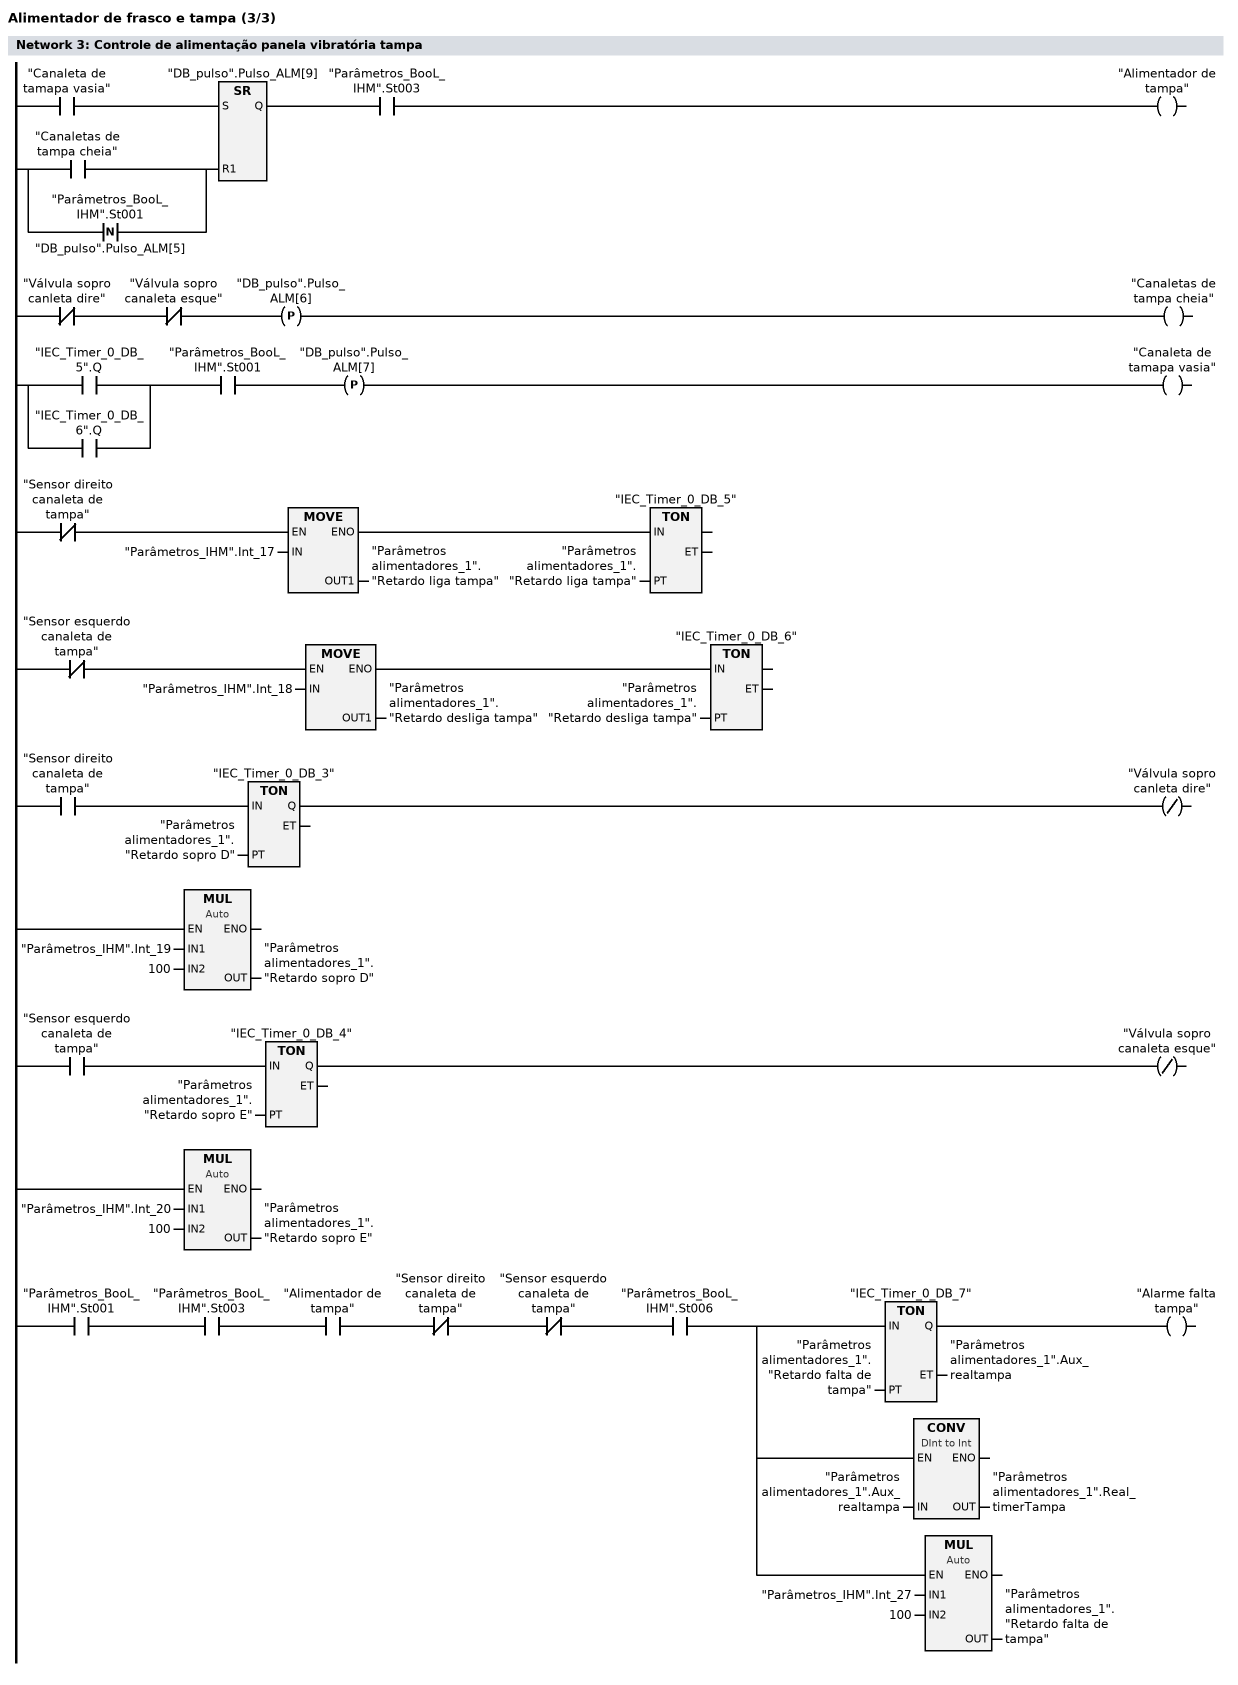
   #_w1 := NOT "Parâmetros_BooL_IHM".St001 AND "DB_pulso".Pulso_ALM[5];   // falling edge of "Parâmetros_BooL_IHM".St001
   "DB_pulso".Pulso_ALM[5] := "Parâmetros_BooL_IHM".St001;
   IF "Canaleta de tamapa vasia" THEN
       "DB_pulso".Pulso_ALM[9] := TRUE;   // SR flip-flop
   END_IF;
   IF "Canaletas de tampa cheia" OR #_w1 THEN "DB_pulso".Pulso_ALM[9] := FALSE; END_IF;
   "Alimentador de tampa" := "DB_pulso".Pulso_ALM[9] AND "Parâmetros_BooL_IHM".St003;
   #_w2 := NOT "Válvula sopro canleta dire" AND NOT "Válvula sopro canaleta esque";
   #_w3 := #_w2 AND NOT "DB_pulso".Pulso_ALM[6];   // rising edge
   "DB_pulso".Pulso_ALM[6] := #_w2;
   "Canaletas de tampa cheia" := #_w3;
   #_w4 := ("IEC_Timer_0_DB_5".Q OR "IEC_Timer_0_DB_6".Q) AND "Parâmetros_BooL_IHM".St001;
   #_w5 := #_w4 AND NOT "DB_pulso".Pulso_ALM[7];   // rising edge
   "DB_pulso".Pulso_ALM[7] := #_w4;
   "Canaleta de tamapa vasia" := #_w5;
   #_w6 := NOT "Sensor direito canaleta de tampa";
   IF #_w6 THEN "Parâmetros alimentadores_1"."Retardo liga tampa" := "Parâmetros_IHM".Int_17; END_IF;
   "IEC_Timer_0_DB_5".TON(IN := #_w6, PT := "Parâmetros alimentadores_1"."Retardo liga tampa");
   #_w7 := NOT "Sensor esquerdo canaleta de tampa";
   IF #_w7 THEN "Parâmetros alimentadores_1"."Retardo desliga tampa" := "Parâmetros_IHM".Int_18; END_IF;
   "IEC_Timer_0_DB_6".TON(IN := #_w7, PT := "Parâmetros alimentadores_1"."Retardo desliga tampa");
   "IEC_Timer_0_DB_3".TON(IN := "Sensor direito canaleta de tampa",
                          PT := "Parâmetros alimentadores_1"."Retardo sopro D");
   "Válvula sopro canleta dire" := NOT "IEC_Timer_0_DB_3".Q;
   "Parâmetros alimentadores_1"."Retardo sopro D" := "Parâmetros_IHM".Int_19 * 100;
   "IEC_Timer_0_DB_4".TON(IN := "Sensor esquerdo canaleta de tampa",
                          PT := "Parâmetros alimentadores_1"."Retardo sopro E");
   "Válvula sopro canaleta esque" := NOT "IEC_Timer_0_DB_4".Q;
   "Parâmetros alimentadores_1"."Retardo sopro E" := "Parâmetros_IHM".Int_20 * 100;
   #_w8 := "Parâmetros_BooL_IHM".St001 AND "Parâmetros_BooL_IHM".St003 AND "Alimentador de tampa" AND NOT "Sensor direito canaleta de tampa" AND NOT "Sensor esquerdo canaleta de tampa" AND "Parâmetros_BooL_IHM".St006;
   "IEC_Timer_0_DB_7".TON(IN := #_w8,
                          PT := "Parâmetros alimentadores_1"."Retardo falta de tampa",
                          ET => "Parâmetros alimentadores_1".Aux_realtampa);
   "Alarme falta tampa" := "IEC_Timer_0_DB_7".Q;
   IF #_w8 THEN
       "Parâmetros alimentadores_1".Real_timerTampa := DINT_TO_INT("Parâmetros alimentadores_1".Aux_realtampa);
       "Parâmetros alimentadores_1"."Retardo falta de tampa" := "Parâmetros_IHM".Int_27 * 100;
   END_IF;
END_REGION
END_FUNCTION

FUNCTION "Controle de produção" : Void   // FC7, LAD
{ S7_Optimized_Access := 'TRUE' }
VERSION : 0.1
   VAR_INPUT
      Habilita_contrle : Bool;
      Deslocamento_transmissão : Bool;
      Fim_envase : Bool;
      Sensor_detector : Bool;
      Rejeito : Bool;
   END_VAR
   VAR_OUTPUT
      Portão_rejeito : Bool;
      Pulso_inspeção : Bool;
   END_VAR
   VAR_IN_OUT
      Controle_habilitado : Bool;
      Total_produção : Int;
      Reprovado : Int;
      Peças_boas : Int;
      Setup_lote : Int;
   END_VAR
   VAR_TEMP   // added for the SCL form of the ladder/FBD networks
      _w1 : Bool;
      _w2 : Bool;
   END_VAR
BEGIN

REGION Network 1: Habilita controle de produção
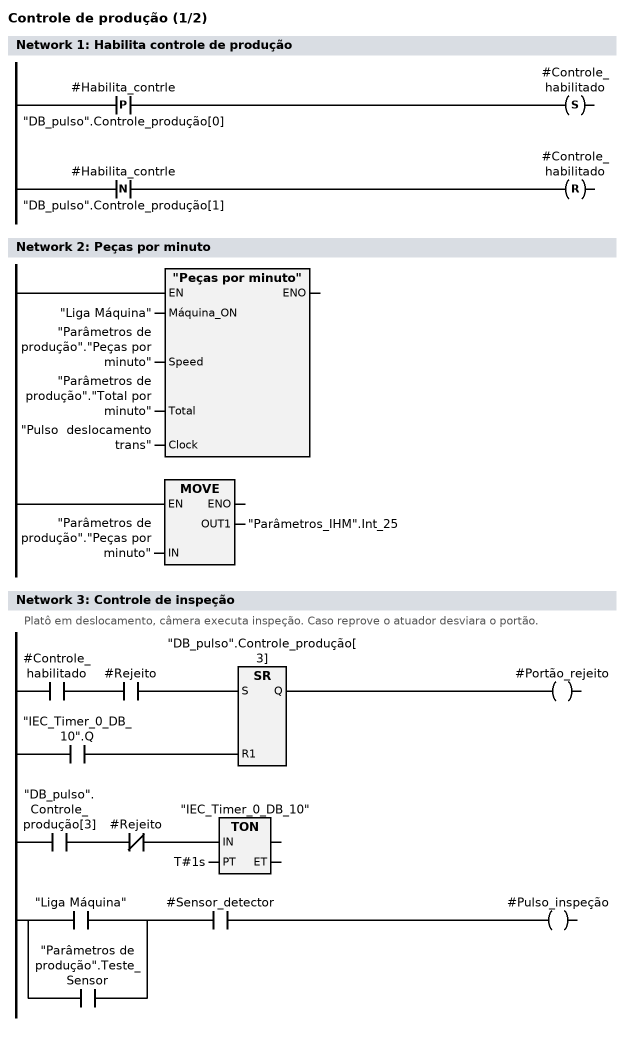
   RUNG wire#powerrail
      P_Contact(operand := #Habilita_contrle, bit := "DB_pulso".Controle_produção[0])
      S_Coil( #Controle_habilitado )
   END_RUNG
   RUNG wire#powerrail
      N_Contact(operand := #Habilita_contrle, bit := "DB_pulso".Controle_produção[1])
      R_Coil( #Controle_habilitado )
   END_RUNG
   // the same network as SCL:
   #_w1 := #Habilita_contrle AND NOT "DB_pulso".Controle_produção[0];   // rising edge of #Habilita_contrle
   "DB_pulso".Controle_produção[0] := #Habilita_contrle;
   IF #_w1 THEN #Controle_habilitado := TRUE; END_IF;
   #_w2 := NOT #Habilita_contrle AND "DB_pulso".Controle_produção[1];   // falling edge of #Habilita_contrle
   "DB_pulso".Controle_produção[1] := #Habilita_contrle;
   IF #_w2 THEN #Controle_habilitado := FALSE; END_IF;
END_REGION

REGION Network 2: Peças por minuto
   RUNG wire#powerrail
      "Peças por minuto"(Máquina_ON := "Liga Máquina", Speed := "Parâmetros de produção"."Peças por minuto", Total := "Parâmetros de produção"."Total por minuto", Clock := "Pulso  deslocamento trans")
   END_RUNG
   RUNG wire#powerrail
      Move(in := "Parâmetros de produção"."Peças por minuto", out1 => "Parâmetros_IHM".Int_25)
   END_RUNG
   // the same network as SCL:
   "Peças por minuto"(Máquina_ON := "Liga Máquina",
                      Speed := "Parâmetros de produção"."Peças por minuto",
                      Total := "Parâmetros de produção"."Total por minuto",
                      Clock := "Pulso  deslocamento trans");
   "Parâmetros_IHM".Int_25 := "Parâmetros de produção"."Peças por minuto";
END_REGION

REGION Network 3: Controle de inspeção
   // Platô em deslocamento, câmera executa inspeção. Caso reprove o atuador desviara o portão.
   IF #Controle_habilitado AND #Rejeito THEN
       "DB_pulso".Controle_produção[3] := TRUE;   // SR flip-flop
   END_IF;
   IF "IEC_Timer_0_DB_10".Q THEN "DB_pulso".Controle_produção[3] := FALSE; END_IF;
   #Portão_rejeito := "DB_pulso".Controle_produção[3];
   "IEC_Timer_0_DB_10".TON(IN := "DB_pulso".Controle_produção[3] AND NOT #Rejeito, PT := T#1s);
   #Pulso_inspeção := ("Liga Máquina" OR "Parâmetros de produção".Teste_Sensor) AND #Sensor_detector;
END_REGION

REGION Network 4: Contagem de produção
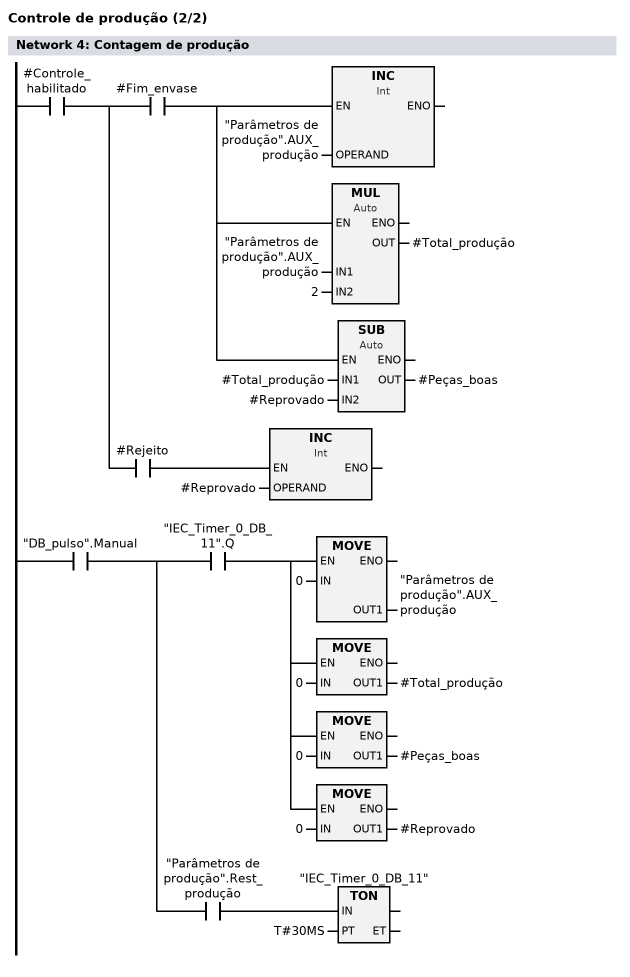
   IF #Controle_habilitado AND #Fim_envase THEN
       "Parâmetros de produção".AUX_produção := "Parâmetros de produção".AUX_produção + 1;
       #Total_produção := "Parâmetros de produção".AUX_produção * 2;
       #Peças_boas := #Total_produção - #Reprovado;
   END_IF;
   IF #Controle_habilitado AND #Rejeito THEN #Reprovado := #Reprovado + 1; END_IF;
   IF "DB_pulso".Manual AND "IEC_Timer_0_DB_11".Q THEN
       "Parâmetros de produção".AUX_produção := 0;
       #Total_produção := 0;
       #Peças_boas := 0;
       #Reprovado := 0;
   END_IF;
   "IEC_Timer_0_DB_11".TON(IN := "DB_pulso".Manual AND "Parâmetros de produção".Rest_produção, PT := T#30MS);
END_REGION
END_FUNCTION

FUNCTION "Alarme" : Void   // FC8, LAD
{ S7_Optimized_Access := 'TRUE' }
VERSION : 0.1
   VAR_OUTPUT
      Restfalahaservodrives : Bool;
      Falha_sincronismo : Bool;
      Atenção : Bool;
   END_VAR
   VAR_IN_OUT
      Status_sincronismo : Bool;
   END_VAR
   VAR_TEMP
      Reset1 : Bool;
      reset2 : Bool;
      reset3 : Bool;
      Status_sincornismo : Bool;
   END_VAR
   VAR_TEMP   // added for the SCL form of the ladder/FBD networks
      _w1 : Bool;
      _w2 : Bool;
      _w3 : Bool;
      _w4 : Bool;
   END_VAR
BEGIN

REGION Network 1: Alarme ativo
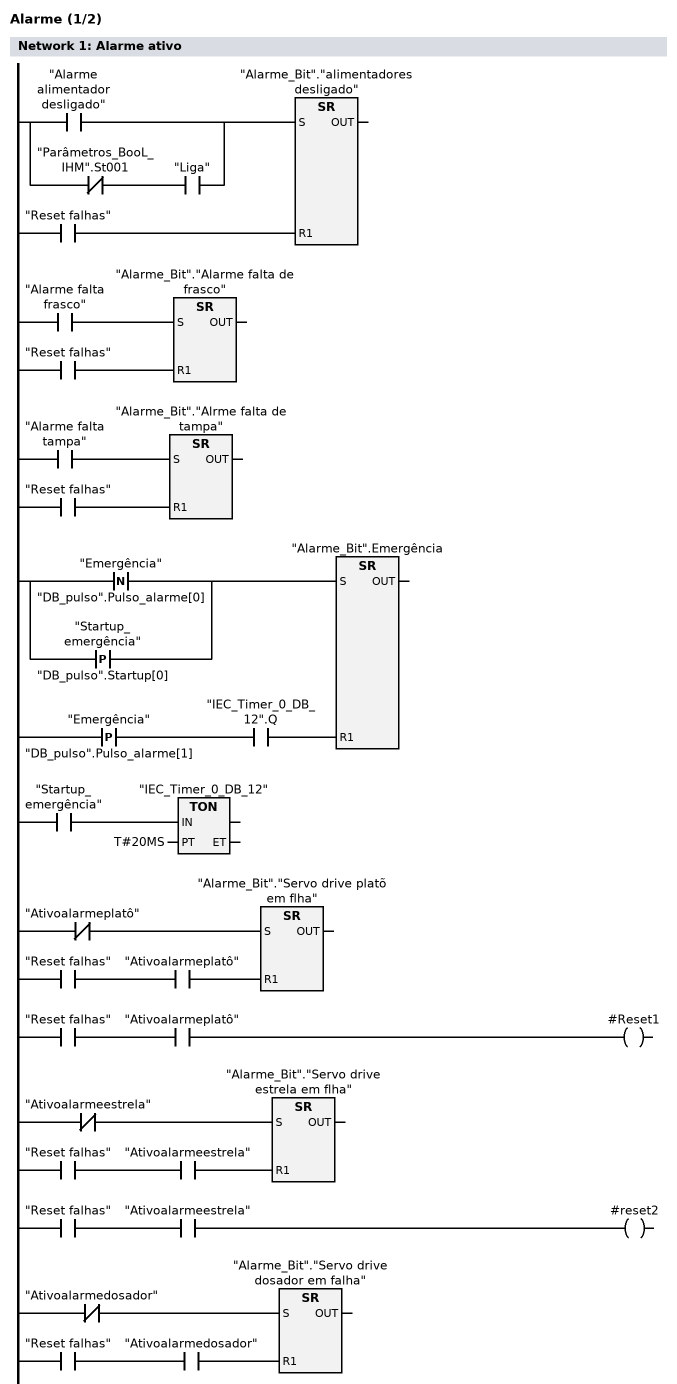
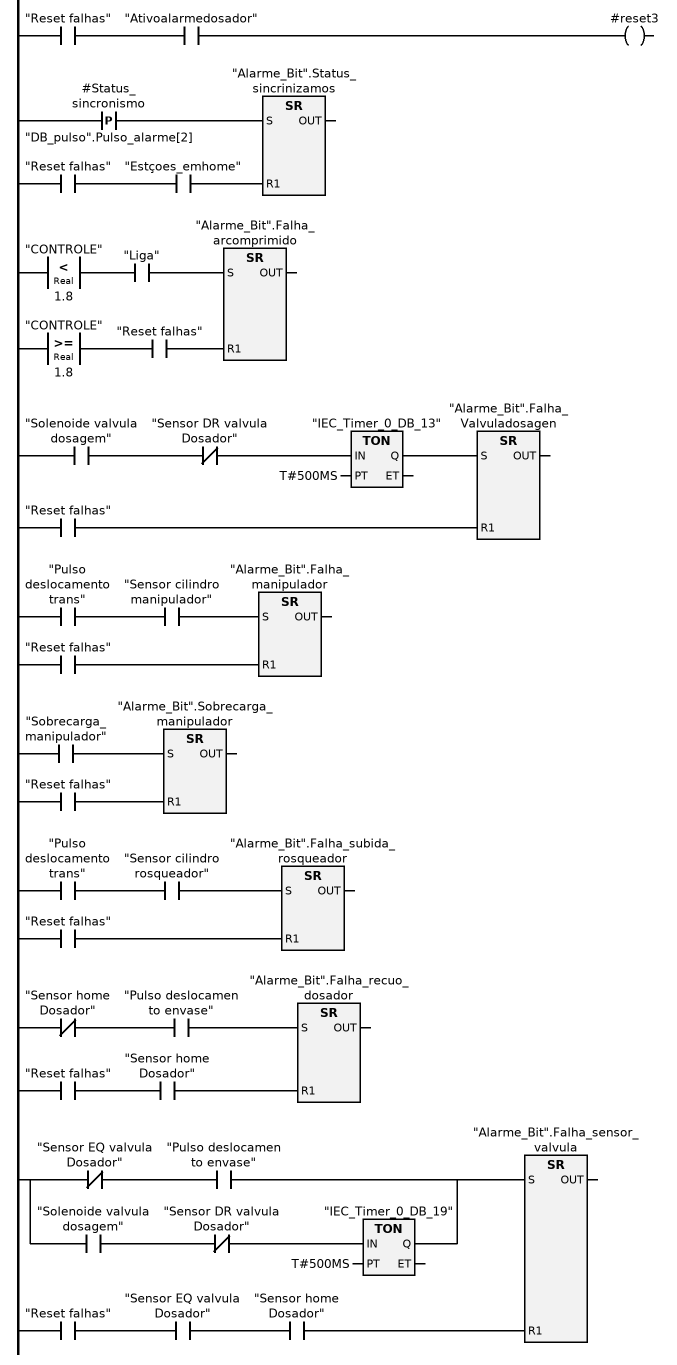
   IF "Alarme alimentador desligado" OR (NOT "Parâmetros_BooL_IHM".St001 AND "Liga") THEN
       "Alarme_Bit"."alimentadores desligado" := TRUE;   // SR flip-flop
   END_IF;
   IF "Reset falhas" THEN "Alarme_Bit"."alimentadores desligado" := FALSE; END_IF;
   IF "Alarme falta frasco" THEN
       "Alarme_Bit"."Alarme falta de frasco" := TRUE;   // SR flip-flop
   END_IF;
   IF "Reset falhas" THEN "Alarme_Bit"."Alarme falta de frasco" := FALSE; END_IF;
   IF "Alarme falta tampa" THEN
       "Alarme_Bit"."Alrme falta de tampa" := TRUE;   // SR flip-flop
   END_IF;
   IF "Reset falhas" THEN "Alarme_Bit"."Alrme falta de tampa" := FALSE; END_IF;
   #_w1 := NOT "Emergência" AND "DB_pulso".Pulso_alarme[0];   // falling edge of "Emergência"
   "DB_pulso".Pulso_alarme[0] := "Emergência";
   #_w2 := "Startup_emergência" AND NOT "DB_pulso".Startup[0];   // rising edge of "Startup_emergência"
   "DB_pulso".Startup[0] := "Startup_emergência";
   #_w3 := "Emergência" AND NOT "DB_pulso".Pulso_alarme[1];   // rising edge of "Emergência"
   "DB_pulso".Pulso_alarme[1] := "Emergência";
   IF #_w1 OR #_w2 THEN
       "Alarme_Bit".Emergência := TRUE;   // SR flip-flop
   END_IF;
   IF #_w3 AND "IEC_Timer_0_DB_12".Q THEN "Alarme_Bit".Emergência := FALSE; END_IF;
   "IEC_Timer_0_DB_12".TON(IN := "Startup_emergência", PT := T#20MS);
   IF NOT "Ativoalarmeplatô" THEN
       "Alarme_Bit"."Servo drive platõ em flha" := TRUE;   // SR flip-flop
   END_IF;
   IF "Reset falhas" AND "Ativoalarmeplatô" THEN "Alarme_Bit"."Servo drive platõ em flha" := FALSE; END_IF;
   #Reset1 := "Reset falhas" AND "Ativoalarmeplatô";
   IF NOT "Ativoalarmeestrela" THEN
       "Alarme_Bit"."Servo drive estrela em flha" := TRUE;   // SR flip-flop
   END_IF;
   IF "Reset falhas" AND "Ativoalarmeestrela" THEN
       "Alarme_Bit"."Servo drive estrela em flha" := FALSE;
   END_IF;
   #reset2 := "Reset falhas" AND "Ativoalarmeestrela";
   IF NOT "Ativoalarmedosador" THEN
       "Alarme_Bit"."Servo drive dosador em falha" := TRUE;   // SR flip-flop
   END_IF;
   IF "Reset falhas" AND "Ativoalarmedosador" THEN
       "Alarme_Bit"."Servo drive dosador em falha" := FALSE;
   END_IF;
   #reset3 := "Reset falhas" AND "Ativoalarmedosador";
   #_w4 := #Status_sincronismo AND NOT "DB_pulso".Pulso_alarme[2];   // rising edge of #Status_sincronismo
   "DB_pulso".Pulso_alarme[2] := #Status_sincronismo;
   IF #_w4 THEN
       "Alarme_Bit".Status_sincrinizamos := TRUE;   // SR flip-flop
   END_IF;
   IF "Reset falhas" AND "Estçoes_emhome" THEN "Alarme_Bit".Status_sincrinizamos := FALSE; END_IF;
   IF ("CONTROLE" < 1.8) AND "Liga" THEN
       "Alarme_Bit".Falha_arcomprimido := TRUE;   // SR flip-flop
   END_IF;
   IF ("CONTROLE" >= 1.8) AND "Reset falhas" THEN "Alarme_Bit".Falha_arcomprimido := FALSE; END_IF;
   "IEC_Timer_0_DB_13".TON(IN := "Solenoide valvula dosagem" AND NOT "Sensor DR valvula Dosador", PT := T#500MS);
   IF "IEC_Timer_0_DB_13".Q THEN
       "Alarme_Bit".Falha_Valvuladosagen := TRUE;   // SR flip-flop
   END_IF;
   IF "Reset falhas" THEN "Alarme_Bit".Falha_Valvuladosagen := FALSE; END_IF;
   IF "Pulso  deslocamento trans" AND "Sensor cilindro manipulador" THEN
       "Alarme_Bit".Falha_manipulador := TRUE;   // SR flip-flop
   END_IF;
   IF "Reset falhas" THEN "Alarme_Bit".Falha_manipulador := FALSE; END_IF;
   IF "Sobrecarga_manipulador" THEN
       "Alarme_Bit".Sobrecarga_manipulador := TRUE;   // SR flip-flop
   END_IF;
   IF "Reset falhas" THEN "Alarme_Bit".Sobrecarga_manipulador := FALSE; END_IF;
   IF "Pulso  deslocamento trans" AND "Sensor cilindro rosqueador" THEN
       "Alarme_Bit".Falha_subida_rosqueador := TRUE;   // SR flip-flop
   END_IF;
   IF "Reset falhas" THEN "Alarme_Bit".Falha_subida_rosqueador := FALSE; END_IF;
   IF NOT "Sensor home Dosador" AND "Pulso deslocamento envase" THEN
       "Alarme_Bit".Falha_recuo_dosador := TRUE;   // SR flip-flop
   END_IF;
   IF "Reset falhas" AND "Sensor home Dosador" THEN "Alarme_Bit".Falha_recuo_dosador := FALSE; END_IF;
   "IEC_Timer_0_DB_19".TON(IN := "Solenoide valvula dosagem" AND NOT "Sensor DR valvula Dosador", PT := T#500MS);
   IF (NOT "Sensor EQ valvula Dosador" AND "Pulso deslocamento envase") OR "IEC_Timer_0_DB_19".Q THEN
       "Alarme_Bit".Falha_sensor_valvula := TRUE;   // SR flip-flop
   END_IF;
   IF "Reset falhas" AND "Sensor EQ valvula Dosador" AND "Sensor home Dosador" THEN
       "Alarme_Bit".Falha_sensor_valvula := FALSE;
   END_IF;
END_REGION

REGION Network 2: Reset alarme servo drives
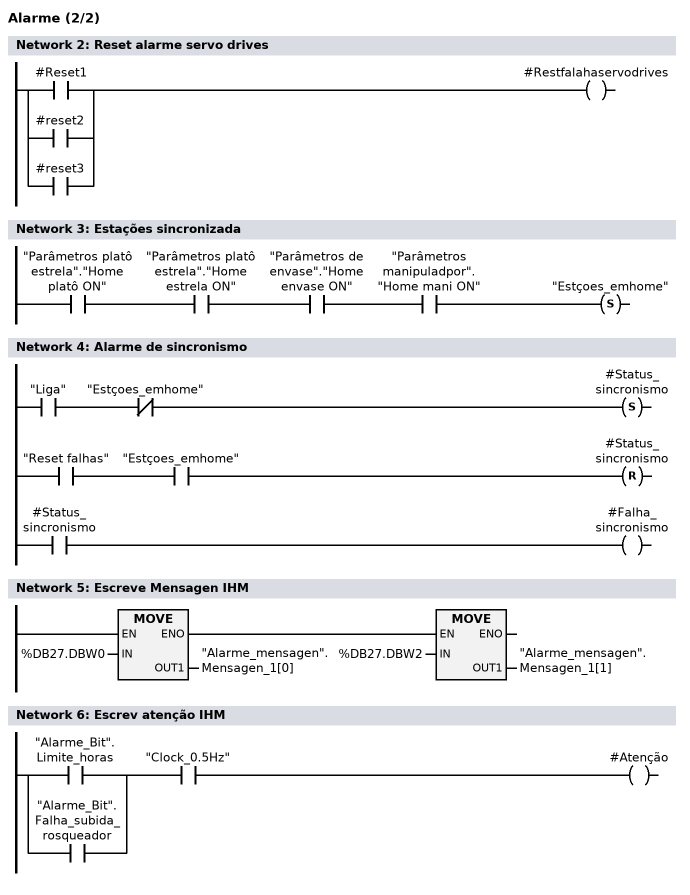
   RUNG wire#powerrail
      Contact( #Reset1 )
      wire#w1
      Coil( #Restfalahaservodrives )
   END_RUNG
   RUNG wire#powerrail
      Contact( #reset2 )
   END_RUNG wire#w1
   RUNG wire#powerrail
      Contact( #reset3 )
   END_RUNG wire#w1
   // the same network as SCL:
   #Restfalahaservodrives := #Reset1 OR #reset2 OR #reset3;
END_REGION

REGION Network 3: Estações sincronizada
   RUNG wire#powerrail
      Contact( "Parâmetros platô estrela"."Home platô ON" )
      Contact( "Parâmetros platô estrela"."Home estrela ON" )
      Contact( "Parâmetros de envase"."Home envase ON" )
      Contact( "Parâmetros manipuladpor"."Home mani ON" )
      S_Coil( "Estçoes_emhome" )
   END_RUNG
   // the same network as SCL:
   IF "Parâmetros platô estrela"."Home platô ON" AND "Parâmetros platô estrela"."Home estrela ON" AND "Parâmetros de envase"."Home envase ON" AND "Parâmetros manipuladpor"."Home mani ON" THEN
       "Estçoes_emhome" := TRUE;
   END_IF;
END_REGION

REGION Network 4: Alarme de sincronismo
   RUNG wire#powerrail
      Contact( "Liga" )
      I_Contact( "Estçoes_emhome" )
      S_Coil( #Status_sincronismo )
   END_RUNG
   RUNG wire#powerrail
      Contact( "Reset falhas" )
      Contact( "Estçoes_emhome" )
      R_Coil( #Status_sincronismo )
   END_RUNG
   RUNG wire#powerrail
      Contact( #Status_sincronismo )
      Coil( #Falha_sincronismo )
   END_RUNG
   // the same network as SCL:
   IF "Liga" AND NOT "Estçoes_emhome" THEN #Status_sincronismo := TRUE; END_IF;
   IF "Reset falhas" AND "Estçoes_emhome" THEN #Status_sincronismo := FALSE; END_IF;
   #Falha_sincronismo := #Status_sincronismo;
END_REGION

REGION Network 5: Escreve Mensagen IHM
   RUNG wire#powerrail
      Move(in := %DB27.DBW0, out1 => "Alarme_mensagen".Mensagen_1[0])
      Move(in := %DB27.DBW2, out1 => "Alarme_mensagen".Mensagen_1[1])
   END_RUNG
   // the same network as SCL:
   "Alarme_mensagen".Mensagen_1[0] := %DB27.DBW0;
   "Alarme_mensagen".Mensagen_1[1] := %DB27.DBW2;
END_REGION

REGION Network 6: Escrev atenção IHM
   RUNG wire#powerrail
      Contact( "Alarme_Bit".Limite_horas )
      wire#w1
      Contact( "Clock_0.5Hz" )
      Coil( #Atenção )
   END_RUNG
   RUNG wire#powerrail
      Contact( "Alarme_Bit".Falha_subida_rosqueador )
   END_RUNG wire#w1
   // the same network as SCL:
   #Atenção := ("Alarme_Bit".Limite_horas OR "Alarme_Bit".Falha_subida_rosqueador) AND "Clock_0.5Hz";
END_REGION
END_FUNCTION

FUNCTION "AR Comprimido" : Void   // FC9, LAD
{ S7_Optimized_Access := 'TRUE' }
VERSION : 0.1
BEGIN

REGION Network 1: Leitura de sensor de pressão
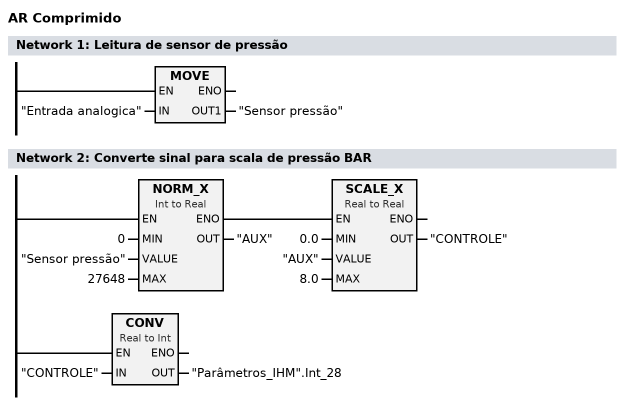
   RUNG wire#powerrail
      Move(in := "Entrada analogica", out1 => "Sensor pressão")
   END_RUNG
   // the same network as SCL:
   "Sensor pressão" := "Entrada analogica";
END_REGION

REGION Network 2: Converte sinal para scala de pressão BAR
   RUNG wire#powerrail
      { S7_Templates := "[SrcType := Int, DestType := Real]" } Normalize(min := 0, value := "Sensor pressão", max := 27648, out => "AUX")
      { S7_Templates := "[SrcType := Real, DestType := Real]" } Scale(min := 0.0, value := "AUX", max := 8.0, out => "CONTROLE")
   END_RUNG
   RUNG wire#powerrail
      { S7_Templates := "[SrcType := Real, DestType := Int]" } Convert(in := "CONTROLE", out => "Parâmetros_IHM".Int_28)
   END_RUNG
   // the same network as SCL:
   "AUX" := NORM_X(MIN := 0, VALUE := "Sensor pressão", MAX := 27648);
   "CONTROLE" := SCALE_X(MIN := 0.0, VALUE := "AUX", MAX := 8.0);
   "Parâmetros_IHM".Int_28 := REAL_TO_INT("CONTROLE");
END_REGION
END_FUNCTION

FUNCTION "Peças por minuto" : Void   // FC10, LAD
{ S7_Optimized_Access := 'TRUE' }
VERSION : 0.1
   VAR_INPUT
      Máquina_ON : Bool;
   END_VAR
   VAR_IN_OUT
      Speed : DInt;
      Total : DInt;
      Clock : Bool;
   END_VAR
BEGIN

REGION Network 1: Contador de peça por minuto
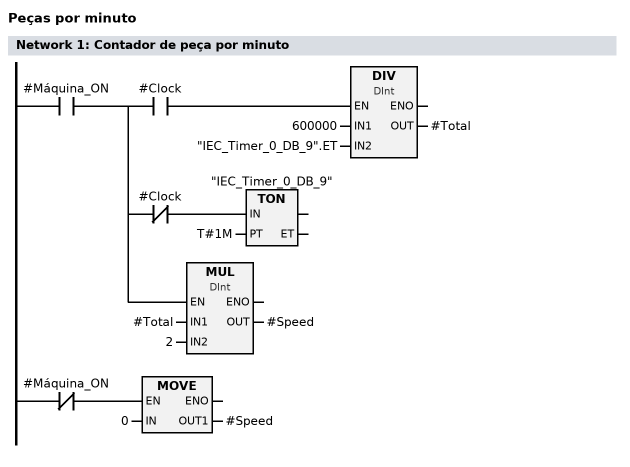
   IF #Máquina_ON AND #Clock THEN #Total := 600000 / "IEC_Timer_0_DB_9".ET; END_IF;
   "IEC_Timer_0_DB_9".TON(IN := #Máquina_ON AND NOT #Clock, PT := T#1M);
   IF #Máquina_ON THEN #Speed := #Total * 2; END_IF;
   IF NOT #Máquina_ON THEN #Speed := 0; END_IF;
END_REGION
END_FUNCTION

FUNCTION "Recipe" : Void   // FC11, LAD
{ S7_Optimized_Access := 'TRUE' }
VERSION : 0.1
   VAR_TEMP   // added for the SCL form of the ladder/FBD networks
      _w1 : Bool;
   END_VAR
BEGIN

REGION Network 1: Download recita
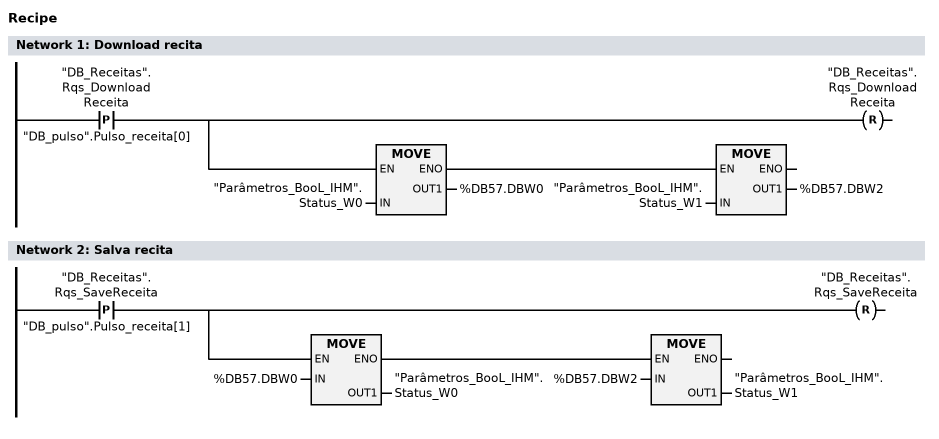
   RUNG wire#powerrail
      P_Contact(operand := "DB_Receitas".Rqs_DownloadReceita, bit := "DB_pulso".Pulso_receita[0])
      wire#w1
      R_Coil( "DB_Receitas".Rqs_DownloadReceita )
   END_RUNG
   RUNG wire#w1
      Move(in := "Parâmetros_BooL_IHM".Status_W0, out1 => %DB57.DBW0)
      Move(in := "Parâmetros_BooL_IHM".Status_W1, out1 => %DB57.DBW2)
   END_RUNG
   // the same network as SCL:
   #_w1 := "DB_Receitas".Rqs_DownloadReceita AND NOT "DB_pulso".Pulso_receita[0];   // rising edge of "DB_Receitas".Rqs_DownloadReceita
   "DB_pulso".Pulso_receita[0] := "DB_Receitas".Rqs_DownloadReceita;
   IF #_w1 THEN
       "DB_Receitas".Rqs_DownloadReceita := FALSE;
       %DB57.DBW0 := "Parâmetros_BooL_IHM".Status_W0;
       %DB57.DBW2 := "Parâmetros_BooL_IHM".Status_W1;
   END_IF;
END_REGION

REGION Network 2: Salva recita
   RUNG wire#powerrail
      P_Contact(operand := "DB_Receitas".Rqs_SaveReceita, bit := "DB_pulso".Pulso_receita[1])
      wire#w1
      R_Coil( "DB_Receitas".Rqs_SaveReceita )
   END_RUNG
   RUNG wire#w1
      Move(in := %DB57.DBW0, out1 => "Parâmetros_BooL_IHM".Status_W0)
      Move(in := %DB57.DBW2, out1 => "Parâmetros_BooL_IHM".Status_W1)
   END_RUNG
   // the same network as SCL:
   #_w1 := "DB_Receitas".Rqs_SaveReceita AND NOT "DB_pulso".Pulso_receita[1];   // rising edge of "DB_Receitas".Rqs_SaveReceita
   "DB_pulso".Pulso_receita[1] := "DB_Receitas".Rqs_SaveReceita;
   IF #_w1 THEN
       "DB_Receitas".Rqs_SaveReceita := FALSE;
       "Parâmetros_BooL_IHM".Status_W0 := %DB57.DBW0;
       "Parâmetros_BooL_IHM".Status_W1 := %DB57.DBW2;
   END_IF;
END_REGION
END_FUNCTION

FUNCTION "Habilita_estações" : Void   // FC12, LAD
{ S7_Optimized_Access := 'TRUE' }
VERSION : 0.1
BEGIN

REGION Network 1: ON OFF estações
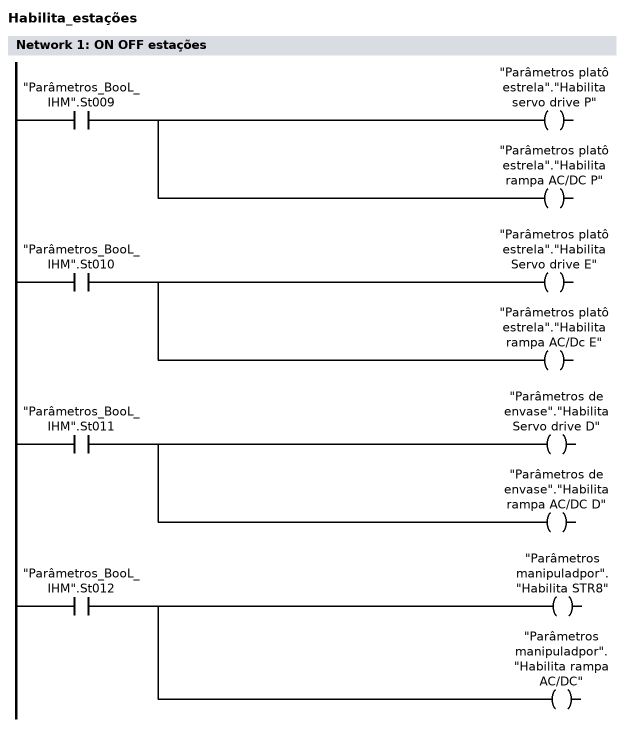
   RUNG wire#powerrail
      Contact( "Parâmetros_BooL_IHM".St009 )
      wire#w1
      Coil( "Parâmetros platô estrela"."Habilita servo drive P" )
   END_RUNG
   RUNG wire#w1
      Coil( "Parâmetros platô estrela"."Habilita rampa AC/DC P" )
   END_RUNG
   RUNG wire#powerrail
      Contact( "Parâmetros_BooL_IHM".St010 )
      wire#w2
      Coil( "Parâmetros platô estrela"."Habilita Servo drive E" )
   END_RUNG
   RUNG wire#w2
      Coil( "Parâmetros platô estrela"."Habilita rampa AC/Dc E" )
   END_RUNG
   RUNG wire#powerrail
      Contact( "Parâmetros_BooL_IHM".St011 )
      wire#w3
      Coil( "Parâmetros de envase"."Habilita Servo drive D" )
   END_RUNG
   RUNG wire#w3
      Coil( "Parâmetros de envase"."Habilita rampa AC/DC D" )
   END_RUNG
   RUNG wire#powerrail
      Contact( "Parâmetros_BooL_IHM".St012 )
      wire#w4
      Coil( "Parâmetros manipuladpor"."Habilita STR8" )
   END_RUNG
   RUNG wire#w4
      Coil( "Parâmetros manipuladpor"."Habilita rampa AC/DC" )
   END_RUNG
   // the same network as SCL:
   "Parâmetros platô estrela"."Habilita servo drive P" := "Parâmetros_BooL_IHM".St009;
   "Parâmetros platô estrela"."Habilita rampa AC/DC P" := "Parâmetros_BooL_IHM".St009;
   "Parâmetros platô estrela"."Habilita Servo drive E" := "Parâmetros_BooL_IHM".St010;
   "Parâmetros platô estrela"."Habilita rampa AC/Dc E" := "Parâmetros_BooL_IHM".St010;
   "Parâmetros de envase"."Habilita Servo drive D" := "Parâmetros_BooL_IHM".St011;
   "Parâmetros de envase"."Habilita rampa AC/DC D" := "Parâmetros_BooL_IHM".St011;
   "Parâmetros manipuladpor"."Habilita STR8" := "Parâmetros_BooL_IHM".St012;
   "Parâmetros manipuladpor"."Habilita rampa AC/DC" := "Parâmetros_BooL_IHM".St012;
END_REGION
END_FUNCTION

ORGANIZATION_BLOCK "Main"   // OB1, LAD, ProgramCycle
TITLE = "Main Program Sweep (Cycle)"
{ S7_Optimized_Access := 'TRUE' }
VERSION : 0.1
   VAR_INPUT
      Initial_Call : Bool;   // Initial call of this OB
      Remanence : Bool;   // =True, if remanent data are available
   END_VAR
   VAR_TEMP   // added for the SCL form of the ladder/FBD networks
      _w1 : Bool;
      _w2 : Bool;
      _w3 : Bool;
   END_VAR
BEGIN

REGION Network 1: Liga máquina
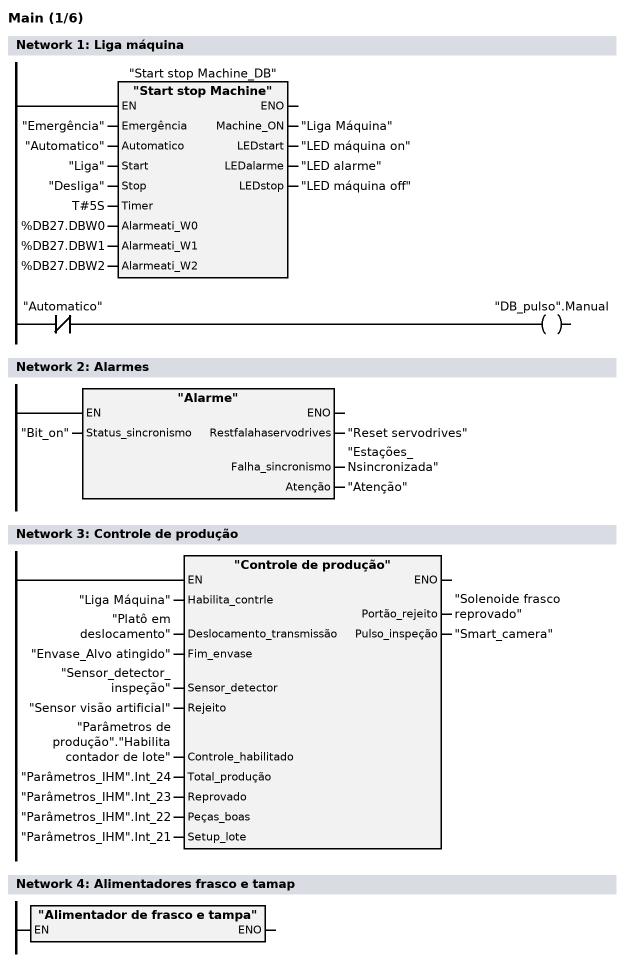
   RUNG wire#powerrail
      "Start stop Machine_DB"(Emergência := "Emergência", Automatico := "Automatico", Start := "Liga", Stop := "Desliga", "Timer" := T#5S, Alarmeati_W0 := %DB27.DBW0, Alarmeati_W1 := %DB27.DBW1, Alarmeati_W2 := %DB27.DBW2, Machine_ON => "Liga Máquina", LEDstart => "LED máquina on", LEDalarme => "LED alarme", LEDstop => "LED máquina off")
   END_RUNG
   RUNG wire#powerrail
      I_Contact( "Automatico" )
      Coil( "DB_pulso".Manual )
   END_RUNG
   // the same network as SCL:
   "Start stop Machine_DB"(Emergência := "Emergência",   // "Start stop Machine"
                           Automatico := "Automatico",
                           Start := "Liga",
                           Stop := "Desliga",
                           "Timer" := T#5S,
                           Alarmeati_W0 := %DB27.DBW0,
                           Alarmeati_W1 := %DB27.DBW1,
                           Alarmeati_W2 := %DB27.DBW2,
                           Machine_ON => "Liga Máquina",
                           LEDstart => "LED máquina on",
                           LEDalarme => "LED alarme",
                           LEDstop => "LED máquina off");
   "DB_pulso".Manual := NOT "Automatico";
END_REGION

REGION Network 2: Alarmes
   RUNG wire#powerrail
      "Alarme"(Status_sincronismo := "Bit_on", Restfalahaservodrives => "Reset servodrives", Falha_sincronismo => "Estações_Nsincronizada", Atenção => "Atenção")
   END_RUNG
   // the same network as SCL:
   "Alarme"(Status_sincronismo := "Bit_on",
            Restfalahaservodrives => "Reset servodrives",
            Falha_sincronismo => "Estações_Nsincronizada",
            Atenção => "Atenção");
END_REGION

REGION Network 3: Controle de produção
   RUNG wire#powerrail
      "Controle de produção"(Habilita_contrle := "Liga Máquina", Deslocamento_transmissão := "Platô em deslocamento", Fim_envase := "Envase_Alvo atingido", Sensor_detector := "Sensor_detector_inspeção", Rejeito := "Sensor visão artificial", Controle_habilitado := "Parâmetros de produção"."Habilita contador de lote", Total_produção := "Parâmetros_IHM".Int_24, Reprovado := "Parâmetros_IHM".Int_23, Peças_boas := "Parâmetros_IHM".Int_22, Setup_lote := "Parâmetros_IHM".Int_21, Portão_rejeito => "Solenoide frasco reprovado", Pulso_inspeção => "Smart_camera")
   END_RUNG
   // the same network as SCL:
   "Controle de produção"(Habilita_contrle := "Liga Máquina",
                          Deslocamento_transmissão := "Platô em deslocamento",
                          Fim_envase := "Envase_Alvo atingido",
                          Sensor_detector := "Sensor_detector_inspeção",
                          Rejeito := "Sensor visão artificial",
                          Controle_habilitado := "Parâmetros de produção"."Habilita contador de lote",
                          Total_produção := "Parâmetros_IHM".Int_24,
                          Reprovado := "Parâmetros_IHM".Int_23,
                          Peças_boas := "Parâmetros_IHM".Int_22,
                          Setup_lote := "Parâmetros_IHM".Int_21,
                          Portão_rejeito => "Solenoide frasco reprovado",
                          Pulso_inspeção => "Smart_camera");
END_REGION

REGION Network 4: Alimentadores frasco e tamap
   RUNG wire#powerrail
      "Alimentador de frasco e tampa"()
   END_RUNG
   // the same network as SCL:
   "Alimentador de frasco e tampa"();
END_REGION

REGION Network 5: Transmissão Plato e estrela
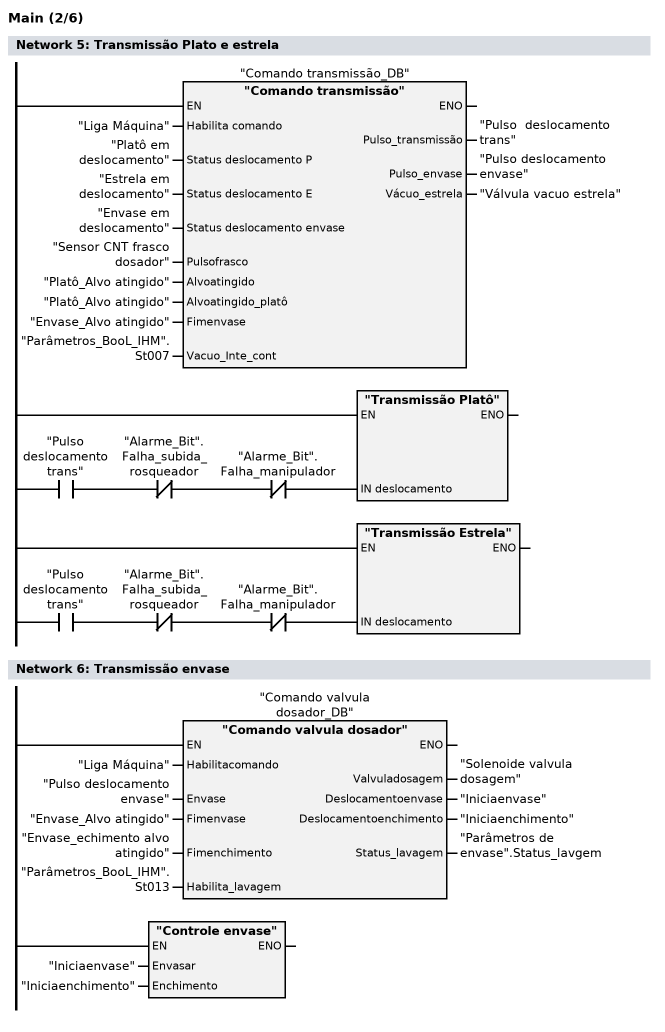
   RUNG wire#powerrail
      "Comando transmissão_DB"("Habilita comando" := "Liga Máquina", "Status deslocamento P" := "Platô em deslocamento", "Status deslocamento E" := "Estrela em deslocamento", "Status deslocamento envase" := "Envase em deslocamento", Pulsofrasco := "Sensor CNT frasco dosador", Alvoatingido := "Platô_Alvo atingido", Alvoatingido_platô := "Platô_Alvo atingido", Fimenvase := "Envase_Alvo atingido", Vacuo_Inte_cont := "Parâmetros_BooL_IHM".St007, Pulso_transmissão => "Pulso  deslocamento trans", Pulso_envase => "Pulso deslocamento envase", Vácuo_estrela => "Válvula vacuo estrela")
   END_RUNG
   RUNG wire#powerrail
      "Transmissão Platô"("IN deslocamento" := wire#w1)
   END_RUNG
   RUNG wire#powerrail
      Contact( "Pulso  deslocamento trans" )
      I_Contact( "Alarme_Bit".Falha_subida_rosqueador )
      I_Contact( "Alarme_Bit".Falha_manipulador )
   END_RUNG wire#w1
   RUNG wire#powerrail
      "Transmissão Estrela"("IN deslocamento" := wire#w2)
   END_RUNG
   RUNG wire#powerrail
      Contact( "Pulso  deslocamento trans" )
      I_Contact( "Alarme_Bit".Falha_subida_rosqueador )
      I_Contact( "Alarme_Bit".Falha_manipulador )
   END_RUNG wire#w2
   // the same network as SCL:
   "Comando transmissão_DB"("Habilita comando" := "Liga Máquina",   // "Comando transmissão"
                           "Status deslocamento P" := "Platô em deslocamento",
                           "Status deslocamento E" := "Estrela em deslocamento",
                           "Status deslocamento envase" := "Envase em deslocamento",
                           Pulsofrasco := "Sensor CNT frasco dosador",
                           Alvoatingido := "Platô_Alvo atingido",
                           Alvoatingido_platô := "Platô_Alvo atingido",
                           Fimenvase := "Envase_Alvo atingido",
                           Vacuo_Inte_cont := "Parâmetros_BooL_IHM".St007,
                           Pulso_transmissão => "Pulso  deslocamento trans",
                           Pulso_envase => "Pulso deslocamento envase",
                           Vácuo_estrela => "Válvula vacuo estrela");
   "Transmissão Platô"("IN deslocamento" := "Pulso  deslocamento trans" AND NOT "Alarme_Bit".Falha_subida_rosqueador AND NOT "Alarme_Bit".Falha_manipulador);
   "Transmissão Estrela"("IN deslocamento" := "Pulso  deslocamento trans" AND NOT "Alarme_Bit".Falha_subida_rosqueador AND NOT "Alarme_Bit".Falha_manipulador);
END_REGION

REGION Network 6: Transmissão envase
   RUNG wire#powerrail
      "Comando valvula dosador_DB"(Habilitacomando := "Liga Máquina", Envase := "Pulso deslocamento envase", Fimenvase := "Envase_Alvo atingido", Fimenchimento := "Envase_echimento alvo atingido", Habilita_lavagem := "Parâmetros_BooL_IHM".St013, Valvuladosagem => "Solenoide valvula dosagem", Deslocamentoenvase => "Iniciaenvase", Deslocamentoenchimento => "Iniciaenchimento", Status_lavagem => "Parâmetros de envase".Status_lavgem)
   END_RUNG
   RUNG wire#powerrail
      "Controle envase"(Envasar := "Iniciaenvase", Enchimento := "Iniciaenchimento")
   END_RUNG
   // the same network as SCL:
   "Comando valvula dosador_DB"(Habilitacomando := "Liga Máquina",   // "Comando valvula dosador"
                           Envase := "Pulso deslocamento envase",
                           Fimenvase := "Envase_Alvo atingido",
                           Fimenchimento := "Envase_echimento alvo atingido",
                           Habilita_lavagem := "Parâmetros_BooL_IHM".St013,
                           Valvuladosagem => "Solenoide valvula dosagem",
                           Deslocamentoenvase => "Iniciaenvase",
                           Deslocamentoenchimento => "Iniciaenchimento",
                           Status_lavagem => "Parâmetros de envase".Status_lavgem);
   "Controle envase"(Envasar := "Iniciaenvase", Enchimento := "Iniciaenchimento");
END_REGION

REGION Network 7: Transmissão Manipulador
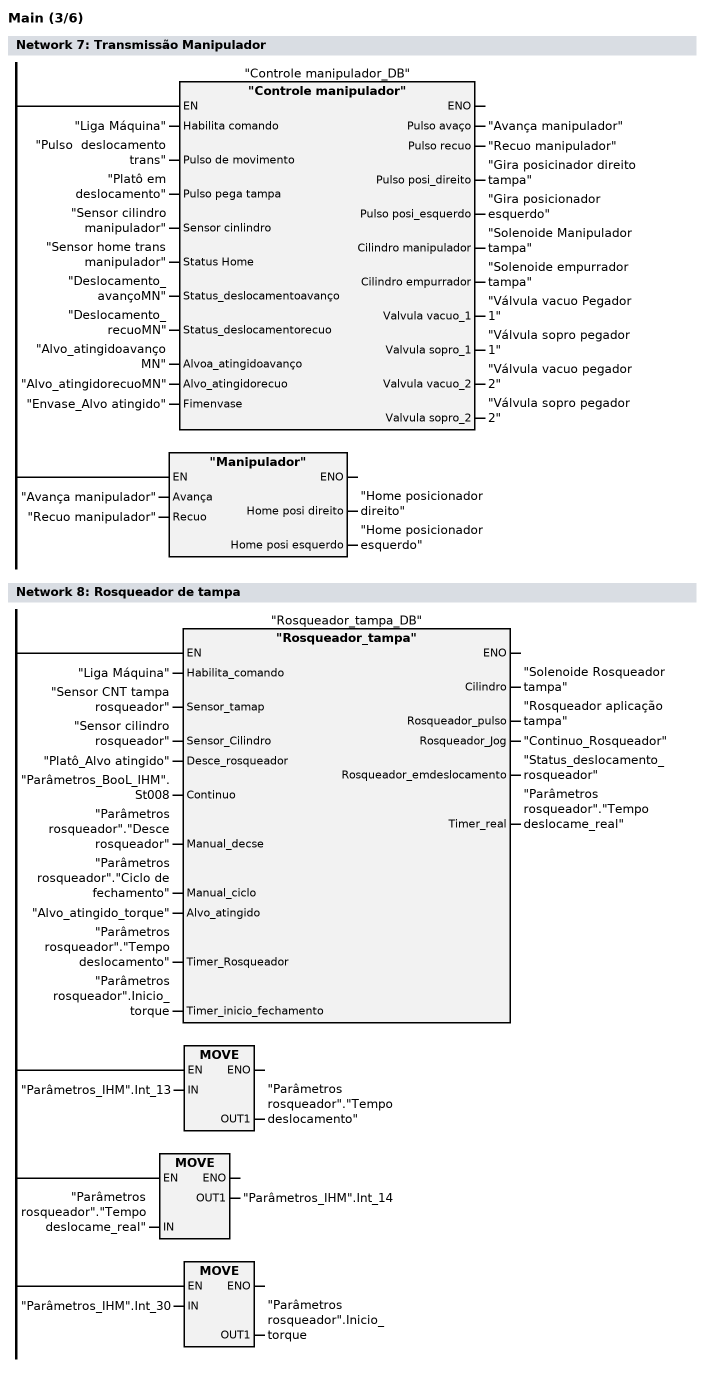
   RUNG wire#powerrail
      "Controle manipulador_DB"("Habilita comando" := "Liga Máquina", "Pulso de movimento" := "Pulso  deslocamento trans", "Pulso pega tampa" := "Platô em deslocamento", "Sensor cinlindro" := "Sensor cilindro manipulador", "Status Home" := "Sensor home trans manipulador", Status_deslocamentoavanço := "Deslocamento_avançoMN", Status_deslocamentorecuo := "Deslocamento_recuoMN", Alvoa_atingidoavanço := "Alvo_atingidoavançoMN", Alvo_atingidorecuo := "Alvo_atingidorecuoMN", Fimenvase := "Envase_Alvo atingido", "Pulso avaço" => "Avança manipulador", "Pulso recuo" => "Recuo manipulador", "Pulso posi_direito" => "Gira posicinador direito tampa", "Pulso posi_esquerdo" => "Gira posicionador esquerdo", "Cilindro manipulador" => "Solenoide Manipulador tampa", "Cilindro empurrador" => "Solenoide empurrador tampa", "Valvula vacuo_1" => "Válvula vacuo Pegador 1", "Valvula sopro_1" => "Válvula sopro pegador 1", "Valvula vacuo_2" => "Válvula vacuo pegador 2", "Valvula sopro_2" => "Válvula sopro pegador 2")
   END_RUNG
   RUNG wire#powerrail
      "Manipulador"(Avança := "Avança manipulador", Recuo := "Recuo manipulador", "Home posi direito" => "Home posicionador direito", "Home posi esquerdo" => "Home posicionador esquerdo")
   END_RUNG
   // the same network as SCL:
   "Controle manipulador_DB"("Habilita comando" := "Liga Máquina",   // "Controle manipulador"
                           "Pulso de movimento" := "Pulso  deslocamento trans",
                           "Pulso pega tampa" := "Platô em deslocamento",
                           "Sensor cinlindro" := "Sensor cilindro manipulador",
                           "Status Home" := "Sensor home trans manipulador",
                           Status_deslocamentoavanço := "Deslocamento_avançoMN",
                           Status_deslocamentorecuo := "Deslocamento_recuoMN",
                           Alvoa_atingidoavanço := "Alvo_atingidoavançoMN",
                           Alvo_atingidorecuo := "Alvo_atingidorecuoMN",
                           Fimenvase := "Envase_Alvo atingido",
                           "Pulso avaço" => "Avança manipulador",
                           "Pulso recuo" => "Recuo manipulador",
                           "Pulso posi_direito" => "Gira posicinador direito tampa",
                           "Pulso posi_esquerdo" => "Gira posicionador esquerdo",
                           "Cilindro manipulador" => "Solenoide Manipulador tampa",
                           "Cilindro empurrador" => "Solenoide empurrador tampa",
                           "Valvula vacuo_1" => "Válvula vacuo Pegador 1",
                           "Valvula sopro_1" => "Válvula sopro pegador 1",
                           "Valvula vacuo_2" => "Válvula vacuo pegador 2",
                           "Valvula sopro_2" => "Válvula sopro pegador 2");
   "Manipulador"(Avança := "Avança manipulador",
                 Recuo := "Recuo manipulador",
                 "Home posi direito" => "Home posicionador direito",
                 "Home posi esquerdo" => "Home posicionador esquerdo");
END_REGION

REGION Network 8: Rosqueador de tampa
   RUNG wire#powerrail
      "Rosqueador_tampa_DB"(Habilita_comando := "Liga Máquina", Sensor_tamap := "Sensor CNT tampa rosqueador", Sensor_Cilindro := "Sensor cilindro rosqueador", Desce_rosqueador := "Platô_Alvo atingido", Continuo := "Parâmetros_BooL_IHM".St008, Manual_decse := "Parâmetros rosqueador"."Desce rosqueador", Manual_ciclo := "Parâmetros rosqueador"."Ciclo de fechamento", Alvo_atingido := "Alvo_atingido_torque", Timer_Rosqueador := "Parâmetros rosqueador"."Tempo deslocamento", Timer_inicio_fechamento := "Parâmetros rosqueador".Inicio_torque, Cilindro => "Solenoide Rosqueador tampa", Rosqueador_pulso => "Rosqueador aplicação tampa", Rosqueador_Jog => "Continuo_Rosqueador", Rosqueador_emdeslocamento => "Status_deslocamento_rosqueador", Timer_real => "Parâmetros rosqueador"."Tempo deslocame_real")
   END_RUNG
   RUNG wire#powerrail
      Move(in := "Parâmetros_IHM".Int_13, out1 => "Parâmetros rosqueador"."Tempo deslocamento")
   END_RUNG
   RUNG wire#powerrail
      Move(in := "Parâmetros rosqueador"."Tempo deslocame_real", out1 => "Parâmetros_IHM".Int_14)
   END_RUNG
   RUNG wire#powerrail
      Move(in := "Parâmetros_IHM".Int_30, out1 => "Parâmetros rosqueador".Inicio_torque)
   END_RUNG
   // the same network as SCL:
   "Rosqueador_tampa_DB"(Habilita_comando := "Liga Máquina",   // "Rosqueador_tampa"
                         Sensor_tamap := "Sensor CNT tampa rosqueador",
                         Sensor_Cilindro := "Sensor cilindro rosqueador",
                         Desce_rosqueador := "Platô_Alvo atingido",
                         Continuo := "Parâmetros_BooL_IHM".St008,
                         Manual_decse := "Parâmetros rosqueador"."Desce rosqueador",
                         Manual_ciclo := "Parâmetros rosqueador"."Ciclo de fechamento",
                         Alvo_atingido := "Alvo_atingido_torque",
                         Timer_Rosqueador := "Parâmetros rosqueador"."Tempo deslocamento",
                         Timer_inicio_fechamento := "Parâmetros rosqueador".Inicio_torque,
                         Cilindro => "Solenoide Rosqueador tampa",
                         Rosqueador_pulso => "Rosqueador aplicação tampa",
                         Rosqueador_Jog => "Continuo_Rosqueador",
                         Rosqueador_emdeslocamento => "Status_deslocamento_rosqueador",
                         Timer_real => "Parâmetros rosqueador"."Tempo deslocame_real");
   "Parâmetros rosqueador"."Tempo deslocamento" := "Parâmetros_IHM".Int_13;
   "Parâmetros_IHM".Int_14 := "Parâmetros rosqueador"."Tempo deslocame_real";
   "Parâmetros rosqueador".Inicio_torque := "Parâmetros_IHM".Int_30;
END_REGION

REGION Network 9: Controle de AR comprimido
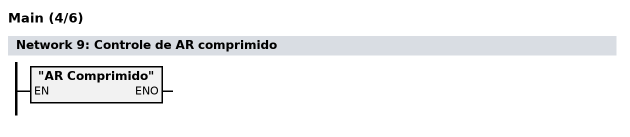
   RUNG wire#powerrail
      "AR Comprimido"()
   END_RUNG
   // the same network as SCL:
   "AR Comprimido"();
END_REGION

REGION Network 10: Clock plc
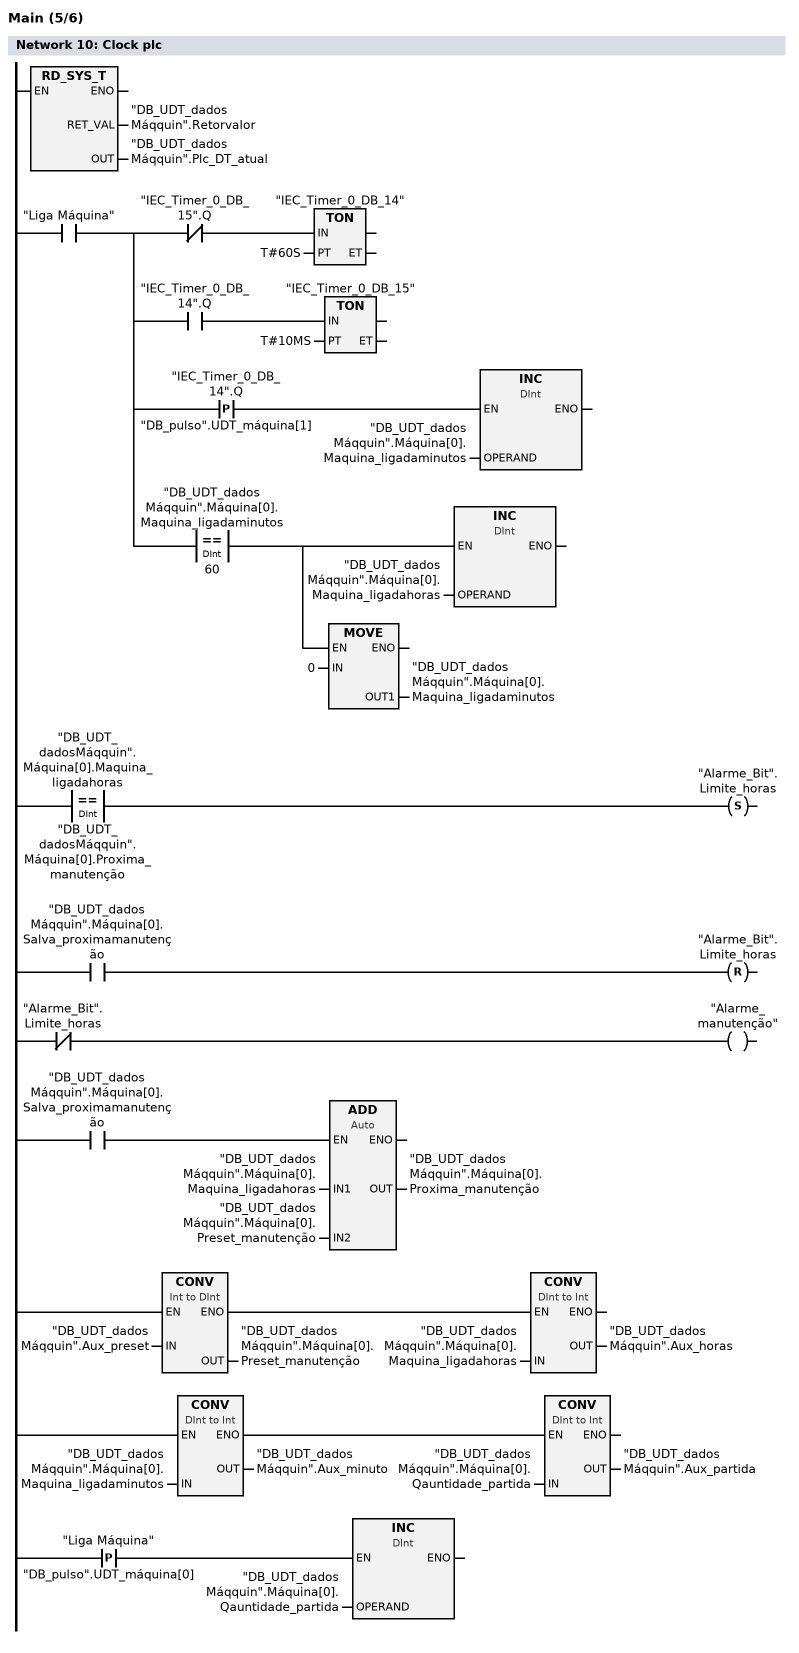
   "DB_UDT_dadosMáqquin".Retorvalor := RD_SYS_T(OUT => "DB_UDT_dadosMáqquin".Plc_DT_atual);
   "IEC_Timer_0_DB_14".TON(IN := "Liga Máquina" AND NOT "IEC_Timer_0_DB_15".Q, PT := T#60S);
   "IEC_Timer_0_DB_15".TON(IN := "Liga Máquina" AND "IEC_Timer_0_DB_14".Q, PT := T#10MS);
   #_w1 := "Liga Máquina" AND "IEC_Timer_0_DB_14".Q AND NOT "DB_pulso".UDT_máquina[1];   // rising edge of "IEC_Timer_0_DB_14".Q
   "DB_pulso".UDT_máquina[1] := "IEC_Timer_0_DB_14".Q;
   IF #_w1 THEN
       "DB_UDT_dadosMáqquin".Máquina[0].Maquina_ligadaminutos := "DB_UDT_dadosMáqquin".Máquina[0].Maquina_ligadaminutos + 1;
   END_IF;
   #_w2 := "Liga Máquina" AND ("DB_UDT_dadosMáqquin".Máquina[0].Maquina_ligadaminutos = 60);
   IF #_w2 THEN
       "DB_UDT_dadosMáqquin".Máquina[0].Maquina_ligadahoras := "DB_UDT_dadosMáqquin".Máquina[0].Maquina_ligadahoras + 1;
       "DB_UDT_dadosMáqquin".Máquina[0].Maquina_ligadaminutos := 0;
   END_IF;
   IF "DB_UDT_dadosMáqquin".Máquina[0].Maquina_ligadahoras = "DB_UDT_dadosMáqquin".Máquina[0].Proxima_manutenção THEN
       "Alarme_Bit".Limite_horas := TRUE;
   END_IF;
   IF "DB_UDT_dadosMáqquin".Máquina[0].Salva_proximamanutenção THEN
       "Alarme_Bit".Limite_horas := FALSE;
   END_IF;
   "Alarme_manutenção" := NOT "Alarme_Bit".Limite_horas;
   IF "DB_UDT_dadosMáqquin".Máquina[0].Salva_proximamanutenção THEN
       "DB_UDT_dadosMáqquin".Máquina[0].Proxima_manutenção := "DB_UDT_dadosMáqquin".Máquina[0].Maquina_ligadahoras + "DB_UDT_dadosMáqquin".Máquina[0].Preset_manutenção;
   END_IF;
   "DB_UDT_dadosMáqquin".Máquina[0].Preset_manutenção := INT_TO_DINT("DB_UDT_dadosMáqquin".Aux_preset);
   "DB_UDT_dadosMáqquin".Aux_horas := DINT_TO_INT("DB_UDT_dadosMáqquin".Máquina[0].Maquina_ligadahoras);
   "DB_UDT_dadosMáqquin".Aux_minuto := DINT_TO_INT("DB_UDT_dadosMáqquin".Máquina[0].Maquina_ligadaminutos);
   "DB_UDT_dadosMáqquin".Aux_partida := DINT_TO_INT("DB_UDT_dadosMáqquin".Máquina[0].Qauntidade_partida);
   #_w3 := "Liga Máquina" AND NOT "DB_pulso".UDT_máquina[0];   // rising edge of "Liga Máquina"
   "DB_pulso".UDT_máquina[0] := "Liga Máquina";
   IF #_w3 THEN
       "DB_UDT_dadosMáqquin".Máquina[0].Qauntidade_partida := "DB_UDT_dadosMáqquin".Máquina[0].Qauntidade_partida + 1;
   END_IF;
END_REGION

REGION Network 11: Receita
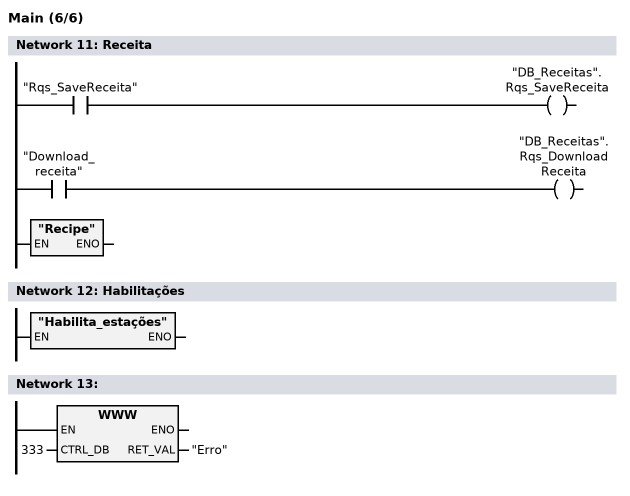
   RUNG wire#powerrail
      Contact( "Rqs_SaveReceita" )
      Coil( "DB_Receitas".Rqs_SaveReceita )
   END_RUNG
   RUNG wire#powerrail
      Contact( "Download_receita" )
      Coil( "DB_Receitas".Rqs_DownloadReceita )
   END_RUNG
   RUNG wire#powerrail
      "Recipe"()
   END_RUNG
   // the same network as SCL:
   "DB_Receitas".Rqs_SaveReceita := "Rqs_SaveReceita";
   "DB_Receitas".Rqs_DownloadReceita := "Download_receita";
   "Recipe"();
END_REGION

REGION Network 12: Habilitações
   RUNG wire#powerrail
      "Habilita_estações"()
   END_RUNG
   // the same network as SCL:
   "Habilita_estações"();
END_REGION

REGION Network 13
   "Erro" := WWW(CTRL_DB := 333);
END_REGION
END_ORGANIZATION_BLOCK

ORGANIZATION_BLOCK "Startup"   // OB100, LAD, Startup
TITLE = "Complete Restart"
{ S7_Optimized_Access := 'TRUE' }
VERSION : 0.1
   VAR_INPUT
      LostRetentive : Bool;   // True if retentive data are lost
      LostRTC : Bool;   // True if date and time are lost
   END_VAR
BEGIN

REGION Network 1: Emrgência
   // Ao energizar a máquina o bit M6.7 vaia a nivel alto levanodo a introção "Alarme_Bit".Emergência ao estador ON.
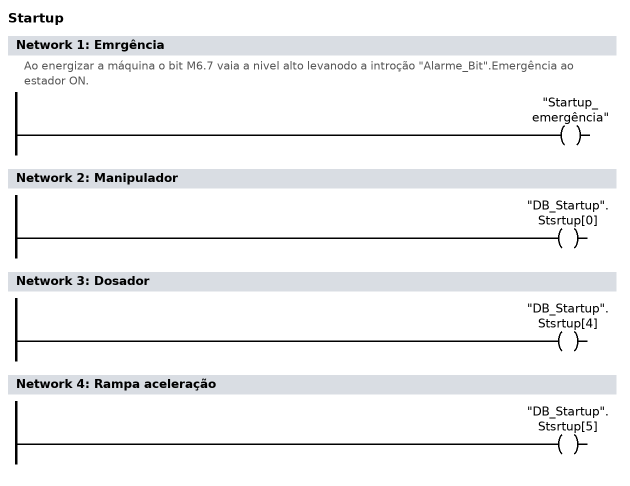
   RUNG wire#powerrail
      Coil( "Startup_emergência" )
   END_RUNG
   // the same network as SCL:
   "Startup_emergência" := TRUE;
END_REGION

REGION Network 2: Manipulador
   RUNG wire#powerrail
      Coil( "DB_Startup".Stsrtup[0] )
   END_RUNG
   // the same network as SCL:
   "DB_Startup".Stsrtup[0] := TRUE;
END_REGION

REGION Network 3: Dosador
   RUNG wire#powerrail
      Coil( "DB_Startup".Stsrtup[4] )
   END_RUNG
   // the same network as SCL:
   "DB_Startup".Stsrtup[4] := TRUE;
END_REGION

REGION Network 4: Rampa aceleração
   RUNG wire#powerrail
      Coil( "DB_Startup".Stsrtup[5] )
   END_RUNG
   // the same network as SCL:
   "DB_Startup".Stsrtup[5] := TRUE;
END_REGION
END_ORGANIZATION_BLOCK